KUKA KRL program: chk_w6_grp7_clo.src

&ACCESS RVO4
&COMMENT Check GRP AXOR Z7 CLOSE
DEF chk_w6_grp7_clo( )

; Check gripper axor CLOSE Z7.1/2
;//---- Start User-------

$TIMER[10] = 0
$TIMER_STOP[10] = FALSE

WAIT FOR (NOT $IN[517] and NOT $in[519])
WAIT FOR ($IN[518] and $in[520])

$TIMER_STOP[10] = TRUE
$TIMER[10] = 0

;//---- End User---------
END
